# EPICS autosave request: ADApp/Db/NDBadPixel_settings.req
$(P)$(R)FileName
file "NDPluginBase_settings.req", P=$(P), R=$(R)
